TYPE ST_Event :
STRUCT
	sDateTime		: STRING;
	sEvent			: STRING;
	fProcVal		: REAL;
	bHeaterState	: BOOL;
END_STRUCT
END_TYPE

(* stored: Version 1.1.0.1, ProductVersion 3.1.4024.3
   DUT ST_Event: Id {10bbdf08-2232-4350-bbc4-f262a5ad1cbc} *)
